{attribute 'qualified_only'}
VAR_GLOBAL
	
	Output_100 AT %i*: ARRAY[0..100] OF Byte;
	Input_100 AT %Q*: ARRAY[0..100] OF Byte;
END_VAR

(* stored: Version 1.1.0.1, ProductVersion 3.1.4024.10
   GVL GVL: Id {1e71d0e2-65e9-4e44-984c-720d3ab1ad3e} *)
